INTERFACE I_MachineLogger

METHOD LogBohrung : BOOL
VAR_INPUT
	stPunkt: REFERENCE TO ST_2DPoint;
END_VAR
END_METHOD

METHOD LogPunktAngefahren : BOOL
VAR_INPUT
	stPunkt: REFERENCE TO ST_2DPoint;
END_VAR
END_METHOD

METHOD LogStart : BOOL
VAR_INPUT
END_VAR
END_METHOD

METHOD LogStop : BOOL
VAR_INPUT
END_VAR
END_METHOD

END_INTERFACE

(* stored: Version 1.1.0.1, ProductVersion 3.1.4024.3
   Itf I_MachineLogger: Id {ea0605d4-5185-4b5d-984f-c3c8fc963e53}
   Method LogBohrung: Id {6f1713fb-3bf1-4926-8549-47014b3f86b1}
   Method LogPunktAngefahren: Id {c428d458-9c9c-440a-9a18-f9a84744d230}
   Method LogStart: Id {d3287210-9333-4d3d-b37c-291ed9128d34}
   Method LogStop: Id {6bdec991-de3f-4ed6-a9cc-3658b807715b} *)
